FUNCTION_BLOCK POU
VAR_INPUT
END_VAR
VAR_OUTPUT
END_VAR
VAR
END_VAR

//Nieuwe POU

END_FUNCTION_BLOCK

(* stored: Version 1.1.0.1, ProductVersion 3.1.4026.8
   POU POU: Id {c4c8e131-3f59-41d1-b7f8-f21eab12f57a}, SpecialFunc None *)
